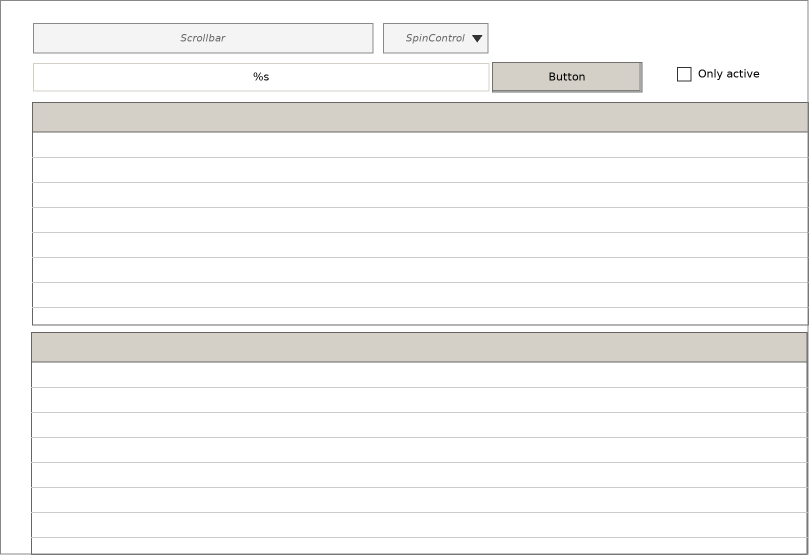
VISUALIZATION Overview  // 809x555
    Button (492,62 150x30), "Button"
        tap MAIN.fbHome.stHmi.bButton
    Table (32,102 777x223), data array: MAIN.fbHome.stHmi.aDigitalIn
        p3854506369: MAIN.fbHome.stHmi.aDigitalIn[INDEX].sName
        p1892666644: MAIN.fbHome.stHmi.aDigitalIn[INDEX].eState
        p338671338: MAIN.fbHome.stHmi.aDigitalIn[INDEX].bValue
    Table (31,332 776x223), data array: MAIN.fbHome.stHmi.aDigitalOut
        p3854506369: MAIN.fbHome.stHmi.aDigitalOut[INDEX].sName
        p1892666644: MAIN.fbHome.stHmi.aDigitalOut[INDEX].eState
        p338671338: MAIN.fbHome.stHmi.aDigitalOut[INDEX].bValue
    SpinControl (383,23 105x30), variable: MAIN.fbHome.stHmi.nInputIndex
        p651134158: MAIN.fbHome.fbDIGroupAll.nSize-1
    Checkbox (675,51 133x46), "Only active", variable: MAIN.fbHome.stHmi.bOnlyActive
    Scrollbar (33,23 340x30)
        p2245068023: MAIN.fbHome.fbDIGroupAll.nSize-1
        p1057716461: MAIN.fbHome.stHmi.nInputIndex
    Textfield (33,63 456x28), "%s", text variable: MAIN.fbHome.stHmi.sInput
END_VISUALIZATION

(* stored: Version 1.1.0.1, ProductVersion 3.1.4024.12
   Visu Overview: Id {5876a2e3-e7ae-4504-b618-e68b8c60ca4d} *)
